// TIA Portal V20 export
DATA_BLOCK "IdentRfInterfaceHmi"   // DB218
// stored: InstanceOfName typeIdentRfHmi, InstanceOfType UDT
"typeIdentRfHmi"
   // VAR
   //    selectedRfReader : USInt;
   //    selectedAntena : USInt;
   //    rfReaderId : USInt;
   //    numberOfRf : USInt;
   //    rfReader : "LSicar_typeIdentInterfaceHmi";
   // END_VAR
BEGIN
END_DATA_BLOCK
